Fanuc KAREL source: kt00002.KL

-- PROVISIONAL review KL for V1013-1; original PC SHA256 3556bd45293af041029ffcf40f550aac004e4b8b05cccd568a3b3b360f642d5f
-- Incomplete behavior may be omitted. Consult companion uncertainty JSON. Do not deploy.
PROGRAM KT00002
%NOLOCKGROUP
VAR
  I1 : INTEGER
  I2 : INTEGER
  OUT : REAL
BEGIN
  -- UNRESOLVED_PC offsets 5-16; opcodes 2E,23
  -- UNRESOLVED_PC offsets 21-32; opcodes 2E,23
  -- UNRESOLVED_PC offsets 37-48; opcodes 2E,23
  -- UNRESOLVED_PC offsets 53-64; opcodes 2E,23
  -- UNRESOLVED_PC offsets 69-89; opcodes 21,21,52,64,23
  -- UNRESOLVED_PC offsets 94-98; opcodes 7F
END KT00002
